  994 = 'S2_Prompts Default 994' | German: 'S2_Prompts German 994' | French: 'S2_Prompts French 994'
  995 = 'S2_Prompts Default 995' | German: 'S2_Prompts German 995' | French: 'S2_Prompts French 995'
  996 = 'S2_Prompts Default 996' | German: 'S2_Prompts German 996' | French: 'S2_Prompts French 996'
  997 = 'S2_Prompts Default 997' | German: 'S2_Prompts German 997' | French: 'S2_Prompts French 997'
  998 = 'S2_Prompts Default 998' | German: 'S2_Prompts German 998' | French: 'S2_Prompts French 998'
  999 = 'S2_Prompts Default 999' | German: 'S2_Prompts German 999' | French: 'S2_Prompts French 999'
  1000 = 'S2_Prompts Default 1000' | German: 'S2_Prompts German 1000' | French: 'S2_Prompts French 1000'
   = ''
END_TEXTLIST

(* stored: Version 1.1.0.1, ProductVersion 3.1.4024.12
   TextList S2_Prompts: Id {07931a1b-3848-4799-af9d-17bab48c96f9} *)
